{attribute 'qualified_only'}
VAR_GLOBAL
	A		: ARRAY[0..CONST.MAX_STATIONS - 1] OF FB_StationA;
	B		: ARRAY[0..CONST.MAX_STATIONS - 1] OF FB_StationB;
END_VAR

(* stored: Version 1.1.0.1
   GVL GVL_Stations: Id {ba5c82c7-e472-49d1-91a6-5ad6132339d1} *)
